TYPE sysTransitions :
STRUCT
    T1 : BOOL;
    T2 : BOOL;
    T3 : BOOL;
    T4 : BOOL;
    T5 : BOOL;
    T6 : BOOL;
    T7 : BOOL;
    T8 : BOOL;
    T9 : BOOL;
    T10 : BOOL;
    T11 : BOOL;
    T12 : BOOL;
    T13 : BOOL;
    T14 : BOOL;
    T15 : BOOL;
    T16 : BOOL;
    T17 : BOOL;
    T18 : BOOL;
    T19 : BOOL;
    T20 : BOOL;
    T21 : BOOL;
    T22 : BOOL;
    T23 : BOOL;
    T24 : BOOL;
    T25 : BOOL;
END_STRUCT
END_TYPE

(* stored: Version 1.1.0.1, ProductVersion 3.1.4026.18
   DUT sysTransitions: Id {de496a14-0215-4043-9689-713acfcac609} *)
